{attribute 'qualified_only'}
VAR_GLOBAL
	ErrAck AT %Q* : BOOL;
	ComErr AT %I* : BOOL;
	EStop AT %I* : BOOL;
END_VAR

(* stored: Version 1.1.0.1, ProductVersion 3.1.4022.18
   GVL SafetyGVL: Id {c6111365-8bce-4b18-a6a1-03511753e6db} *)
